// TwinCAT 3 PLC project MAS418_PLC
// ProgramVersion: 3.1.4023.0
// libraries:
//   Tc2_Standard, * (Beckhoff Automation GmbH)
//   Tc2_System, * (Beckhoff Automation GmbH)
//   Tc3_Module, * (Beckhoff Automation GmbH)
//   VisuDialogs, * (System)
// project tree:
//   / GlobalTextList.TcGTLO, PlcTask.TcTTO, Visualization Manager.TcVMO (not stored)
//   POUs/ HMI.TcVIS, MAIN.TcPOU
// real-time tasks:
//   TASK PlcTask: cycle T#10ms, priority 20, ADS port 350

CONFIGURATION MAS418_PLC
    RESOURCE PLC ON TwinCAT3
        TASK PlcTask(INTERVAL := T#10ms, PRIORITY := 20);
        PROGRAM MAIN WITH PlcTask : MAIN;
    END_RESOURCE
END_CONFIGURATION

// ---- POUs/MAIN.TcPOU
PROGRAM MAIN
VAR
	bEnable : BOOL;
	bStart : BOOL;
	nINT : INT := -32768; 
	nUINT : UINT := 65535;
	fREAL : REAL := 255.255; 
	sPowerStatus: STRING := 'Power Off';
	nFloatConversion : INT; 
	fFloatConversion : LREAL;
END_VAR

bEnable := bStart;
fFloatConversion := INT_TO_REAL(nINT);
nFloatConversion := REAL_TO_INT(fREAL);

END_PROGRAM

// ---- GlobalTextList.TcGTLO
TEXTLIST GlobalTextList
  888 = '%f'
  308 = '%i'
  129 = '%s'
  808 = 'BOOL'
  583 = 'DataTypeTesting'
  497 = 'INT'
  62 = 'Power ON'
  324 = 'REAL'
  612 = 'STRING'
  694 = 'UINT'
END_TEXTLIST

// ---- POUs/HMI.TcVIS
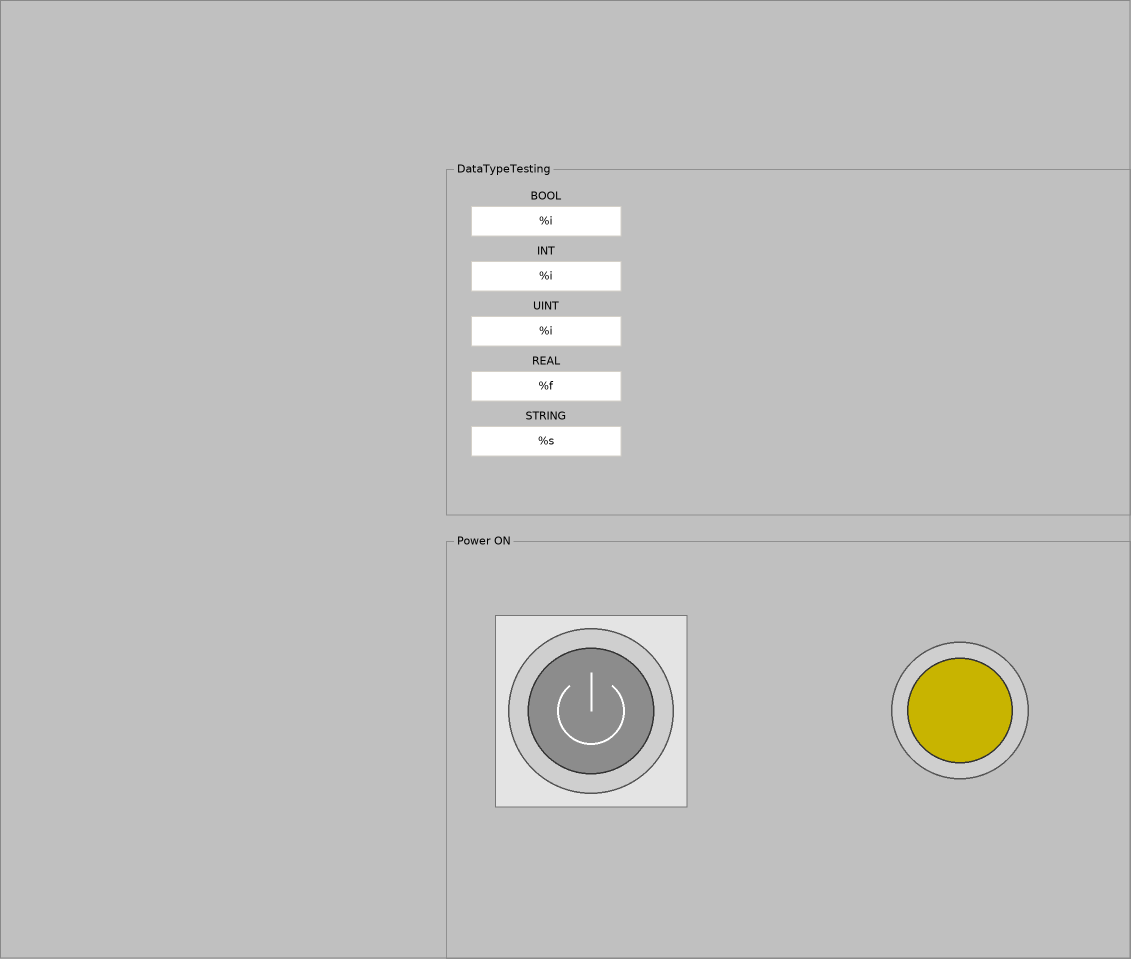
VISUALIZATION HMI  // 1131x959
    GroupBox (446,533 685x426), "Power ON"
        Lamp1 (434,90 160x175), variable: MAIN.bEnable, style: Lamp-Lamp1-Yellow
        PowerSwitch (49,63 192x230), variable: MAIN.bStart, behaviour: TOGGLE, style: Switch-PowerSwitch-Gray
    GroupBox (446,161 685x354), "DataTypeTesting"
        Textfield (25,45 150x30), "%i", text variable: MAIN.bEnable
        Textfield (25,100 150x30), "%i", text variable: MAIN.nINT
        Textfield (25,155 150x30), "%i", text variable: MAIN.nUINT
        Textfield (25,210 150x30), "%f", text variable: MAIN.fREAL
            OnMouseDown: write the text variable via Default
        Textfield (25,265 150x30), "%s", text variable: MAIN.sPowerStatus
            OnMouseDown: write the text variable via Default
        Label (25,20 150x30), "BOOL"
        Label (25,75 150x30), "INT"
        Label (25,130 150x30), "UINT"
        Label (25,185 150x30), "REAL"
        Label (25,240 150x30), "STRING"
END_VISUALIZATION
